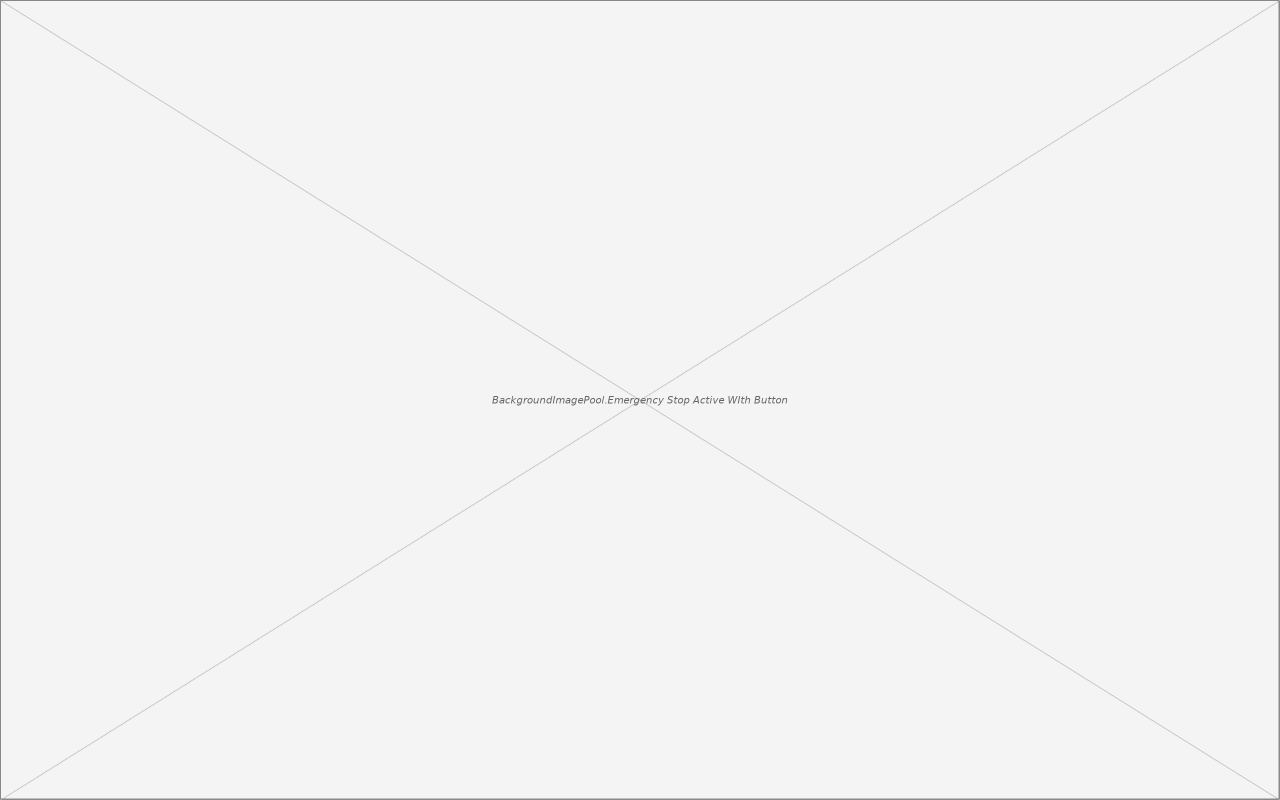
VISUALIZATION Estop  // 1280x800
VAR_IN_OUT
	bHideEstop		: BOOL ; // Hide Estop screen
END_VAR
    Image (0,0 1280x800), invisible if: bHideEstop, input disabled if: bHideEstop, image: BackgroundImagePool.Emergency Stop Active WIth Button
END_VISUALIZATION

(* stored: Version 1.1.0.1, ProductVersion 3.1.4024.5
   Visu Estop: Id {fb475398-f6aa-4891-8c3d-3b6fdd9b8ad0} *)
